// TIA Portal project "水塔水池控制" (V15.1)

(* hardware
DEVICE "S7-1200 station_1"  S7-1200 Station
   slot 0: "Rack_0"  S7-1200 Rack  Rack  V1.0
   slot 1: "PLC_1"  CPU 1214C DC/DC/Rly  6ES7 214-1HG40-0XB0  V4.2
DEVICE "HMI_1"  KTP900 Basic PN
   slot 0: "HMI_1"  KTP900 Basic PN  6AV2 123-2JB03-0AX0  15.1.0.0
   slot 1: "HMI_RT_1"  KTP900 Basic PN  6AV2 123-2JB03-0AX0  15.1.0.0
   slot 5: "HMI_1.IE_CP_1"  PROFINET Interface  15.0.1.0
      slot 1: "PROFINET Interface_1"  PROFINET Interface
         slot 1: "Port_1"  Port
*)

// ===== PLC "PLC_1"  CPU 1214C DC/DC/Rly =====

VAR_GLOBAL   // PLC tag table "默认变量表"
   "S1" AT %M10.0 : Bool;   // 水池下限液位开关
   "S2" AT %M10.1 : Bool;   // 水池上限液位开关
   "S3" AT %M10.2 : Bool;   // 水塔下限液位开关
   "S4" AT %M10.3 : Bool;   // 水塔上限液位开关
   "Start" AT %M10.4 : Bool;
   "Stop" AT %M10.5 : Bool;
   "System_Byte" AT %MB1 : Byte;
   "FirstScan" AT %M1.0 : Bool;
   "DiagStatusUpdate" AT %M1.1 : Bool;
   "AlwaysTRUE" AT %M1.2 : Bool;
   "AlwaysFALSE" AT %M1.3 : Bool;
   "Clock_Byte" AT %MB0 : Byte;
   "Clock_10Hz" AT %M0.0 : Bool;
   "Clock_5Hz" AT %M0.1 : Bool;
   "Clock_2.5Hz" AT %M0.2 : Bool;
   "Clock_2Hz" AT %M0.3 : Bool;
   "Clock_1.25Hz" AT %M0.4 : Bool;
   "Clock_1Hz" AT %M0.5 : Bool;
   "Clock_0.625Hz" AT %M0.6 : Bool;
   "Clock_0.5Hz" AT %M0.7 : Bool;
   "状态0" AT %M2.0 : Bool;
   "状态1" AT %M2.1 : Bool;
   "状态2" AT %M2.2 : Bool;
   "状态3" AT %M2.3 : Bool;
   "状态4" AT %M2.4 : Bool;
   "系统运行状态" AT %M5.0 : Bool;
   "状态5" AT %M2.5 : Bool;
   "Valve" AT %Q0.0 : Bool;
   "Pump" AT %Q0.1 : Bool;
   "Warning" AT %Q0.2 : Bool;
   "水塔状态0" AT %M3.0 : Bool;
   "水塔状态1" AT %M3.1 : Bool;
   "水塔状态2" AT %M3.2 : Bool;
   "水塔状态3" AT %M3.3 : Bool;
   "放水阀" AT %M5.1 : Bool;
   "Byte2" AT %MB2 : Byte;
   "模式选择开关" AT %M5.2 : Bool;
   "Byte3" AT %MB3 : Byte;
   "Tag_1" AT %M5.3 : Bool;
   "手动开阀" AT %M6.0 : Bool;
   "手动启动水泵" AT %M6.1 : Bool;
END_VAR

DATA_BLOCK "HMIdata"   // DB1
{ S7_Optimized_Access := 'TRUE' }
VERSION : 0.1
   VAR
      Tower_water : Int;
      Pool_water : Int;
      Valve_Flow_Num : Int := 10;   // 电磁阀开度
      Pump_Flow_Num : Int := 8;   // 抽水流量大小
      放水阀开度 : Int := 7;   // 放水流量大小
   END_VAR
BEGIN
END_DATA_BLOCK

DATA_BLOCK "水池自动控制_DB"   // DB2
{ S7_Optimized_Access := 'TRUE' }
VERSION : 0.1
// stored: InstanceOfName 水池自动控制
"水池自动控制"
BEGIN
END_DATA_BLOCK

DATA_BLOCK "动画控制_DB"   // DB3
{ S7_Optimized_Access := 'TRUE' }
VERSION : 0.1
// stored: InstanceOfName 动画控制
"动画控制"
BEGIN
END_DATA_BLOCK

DATA_BLOCK "水塔自动控制_DB"   // DB4
{ S7_Optimized_Access := 'TRUE' }
VERSION : 0.1
// stored: InstanceOfName 水塔自动控制
"水塔自动控制"
BEGIN
END_DATA_BLOCK

DATA_BLOCK "手动控制_DB"   // DB5
{ S7_Optimized_Access := 'TRUE' }
VERSION : 0.1
// stored: InstanceOfName 手动控制
"手动控制"
BEGIN
END_DATA_BLOCK

FUNCTION_BLOCK "水池自动控制"   // FB1, LAD
{ S7_Optimized_Access := 'TRUE' }
VERSION : 0.1
   VAR
      T1 : IEC_TIMER;
   END_VAR
   VAR_TEMP   // added for the SCL form of the ladder/FBD networks
      _w1 : Bool;
   END_VAR
BEGIN

REGION Network 1: 初始化
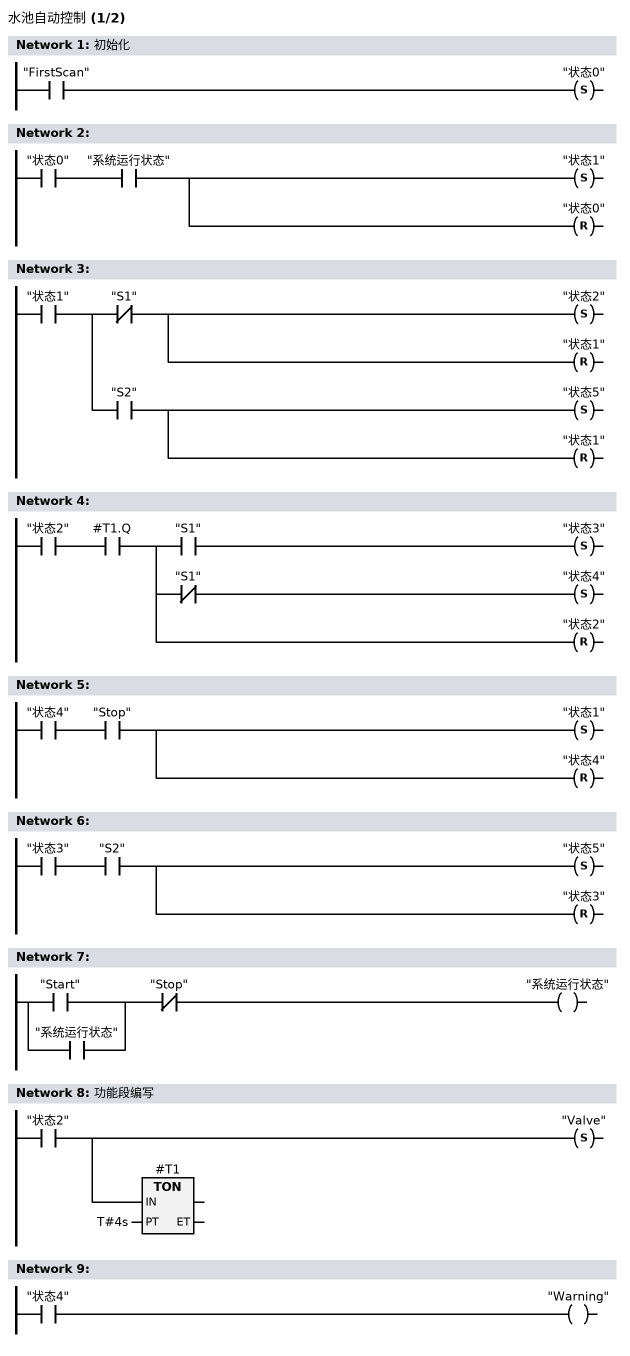
   RUNG wire#powerrail
      Contact( "FirstScan" )
      S_Coil( "状态0" )
   END_RUNG
   // the same network as SCL:
   IF "FirstScan" THEN "状态0" := TRUE; END_IF;
END_REGION

REGION Network 2
   RUNG wire#powerrail
      Contact( "状态0" )
      Contact( "系统运行状态" )
      wire#w1
      S_Coil( "状态1" )
   END_RUNG
   RUNG wire#w1
      R_Coil( "状态0" )
   END_RUNG
   // the same network as SCL:
   IF "状态0" AND "系统运行状态" THEN
       "状态1" := TRUE;
       "状态0" := FALSE;
   END_IF;
END_REGION

REGION Network 3
   RUNG wire#powerrail
      Contact( "状态1" )
      wire#w1
      I_Contact( "S1" )
      wire#w2
      S_Coil( "状态2" )
   END_RUNG
   RUNG wire#w2
      R_Coil( "状态1" )
   END_RUNG
   RUNG wire#w1
      Contact( "S2" )
      wire#w3
      S_Coil( "状态5" )
   END_RUNG
   RUNG wire#w3
      R_Coil( "状态1" )
   END_RUNG
   // the same network as SCL:
   IF "状态1" AND NOT "S1" THEN "状态2" := TRUE; END_IF;
   #_w1 := "状态1";
   IF "状态1" AND NOT "S1" THEN "状态1" := FALSE; END_IF;
   IF #_w1 AND "S2" THEN
       "状态5" := TRUE;
       "状态1" := FALSE;
   END_IF;
END_REGION

REGION Network 4
   RUNG wire#powerrail
      Contact( "状态2" )
      Contact( #T1.Q )
      wire#w1
      Contact( "S1" )
      S_Coil( "状态3" )
   END_RUNG
   RUNG wire#w1
      I_Contact( "S1" )
      S_Coil( "状态4" )
   END_RUNG
   RUNG wire#w1
      R_Coil( "状态2" )
   END_RUNG
   // the same network as SCL:
   #_w1 := "状态2" AND #T1.Q;
   IF #_w1 AND "S1" THEN "状态3" := TRUE; END_IF;
   IF #_w1 AND NOT "S1" THEN "状态4" := TRUE; END_IF;
   IF #_w1 THEN "状态2" := FALSE; END_IF;
END_REGION

REGION Network 5
   RUNG wire#powerrail
      Contact( "状态4" )
      Contact( "Stop" )
      wire#w1
      S_Coil( "状态1" )
   END_RUNG
   RUNG wire#w1
      R_Coil( "状态4" )
   END_RUNG
   // the same network as SCL:
   IF "状态4" AND "Stop" THEN
       "状态1" := TRUE;
       "状态4" := FALSE;
   END_IF;
END_REGION

REGION Network 6
   RUNG wire#powerrail
      Contact( "状态3" )
      Contact( "S2" )
      wire#w1
      S_Coil( "状态5" )
   END_RUNG
   RUNG wire#w1
      R_Coil( "状态3" )
   END_RUNG
   // the same network as SCL:
   IF "状态3" AND "S2" THEN
       "状态5" := TRUE;
       "状态3" := FALSE;
   END_IF;
END_REGION

REGION Network 7
   RUNG wire#powerrail
      Contact( "Start" )
      wire#w1
      I_Contact( "Stop" )
      Coil( "系统运行状态" )
   END_RUNG
   RUNG wire#powerrail
      Contact( "系统运行状态" )
   END_RUNG wire#w1
   // the same network as SCL:
   "系统运行状态" := ("Start" OR "系统运行状态") AND NOT "Stop";
END_REGION

REGION Network 8: 功能段编写
   IF "状态2" THEN "Valve" := TRUE; END_IF;
   #T1.TON(IN := "状态2", PT := T#4s);
END_REGION

REGION Network 9
   RUNG wire#powerrail
      Contact( "状态4" )
      Coil( "Warning" )
   END_RUNG
   // the same network as SCL:
   "Warning" := "状态4";
END_REGION

REGION Network 10
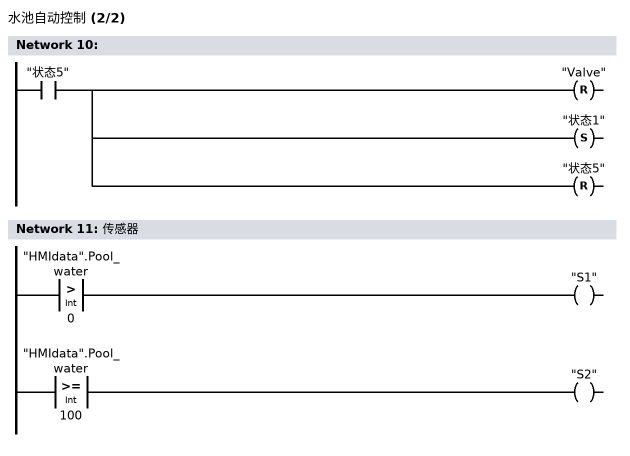
   RUNG wire#powerrail
      Contact( "状态5" )
      wire#w1
      R_Coil( "Valve" )
   END_RUNG
   RUNG wire#w1
      S_Coil( "状态1" )
   END_RUNG
   RUNG wire#w1
      R_Coil( "状态5" )
   END_RUNG
   // the same network as SCL:
   IF "状态5" THEN
       "Valve" := FALSE;
       "状态1" := TRUE;
       "状态5" := FALSE;
   END_IF;
END_REGION

REGION Network 11: 传感器
   RUNG wire#powerrail
      { S7_Templates := "SrcType := Int" } GT_Contact(in1 := "HMIdata".Pool_water, in2 := 0)
      Coil( "S1" )
   END_RUNG
   RUNG wire#powerrail
      { S7_Templates := "SrcType := Int" } GE_Contact(in1 := "HMIdata".Pool_water, in2 := 100)
      Coil( "S2" )
   END_RUNG
   // the same network as SCL:
   "S1" := "HMIdata".Pool_water > 0;
   "S2" := "HMIdata".Pool_water >= 100;
END_REGION
END_FUNCTION_BLOCK

FUNCTION_BLOCK "水塔自动控制"   // FB2, LAD
{ S7_Optimized_Access := 'TRUE' }
VERSION : 0.1
BEGIN

REGION Network 1
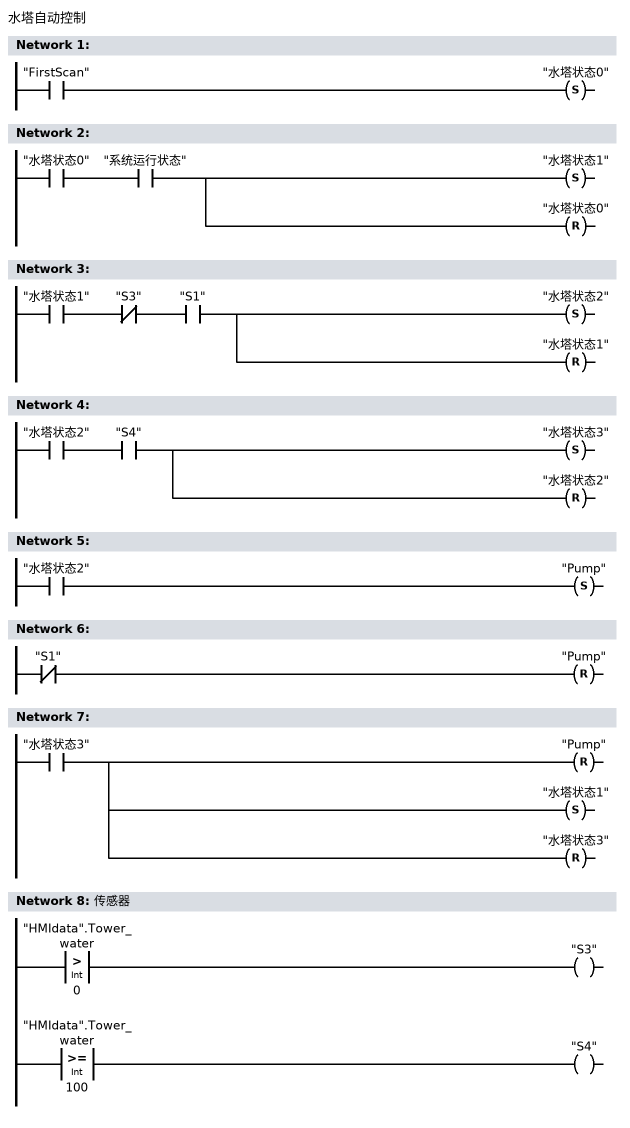
   RUNG wire#powerrail
      Contact( "FirstScan" )
      S_Coil( "水塔状态0" )
   END_RUNG
   // the same network as SCL:
   IF "FirstScan" THEN "水塔状态0" := TRUE; END_IF;
END_REGION

REGION Network 2
   RUNG wire#powerrail
      Contact( "水塔状态0" )
      Contact( "系统运行状态" )
      wire#w1
      S_Coil( "水塔状态1" )
   END_RUNG
   RUNG wire#w1
      R_Coil( "水塔状态0" )
   END_RUNG
   // the same network as SCL:
   IF "水塔状态0" AND "系统运行状态" THEN
       "水塔状态1" := TRUE;
       "水塔状态0" := FALSE;
   END_IF;
END_REGION

REGION Network 3
   RUNG wire#powerrail
      Contact( "水塔状态1" )
      I_Contact( "S3" )
      Contact( "S1" )
      wire#w1
      S_Coil( "水塔状态2" )
   END_RUNG
   RUNG wire#w1
      R_Coil( "水塔状态1" )
   END_RUNG
   // the same network as SCL:
   IF "水塔状态1" AND NOT "S3" AND "S1" THEN
       "水塔状态2" := TRUE;
       "水塔状态1" := FALSE;
   END_IF;
END_REGION

REGION Network 4
   RUNG wire#powerrail
      Contact( "水塔状态2" )
      Contact( "S4" )
      wire#w1
      S_Coil( "水塔状态3" )
   END_RUNG
   RUNG wire#w1
      R_Coil( "水塔状态2" )
   END_RUNG
   // the same network as SCL:
   IF "水塔状态2" AND "S4" THEN
       "水塔状态3" := TRUE;
       "水塔状态2" := FALSE;
   END_IF;
END_REGION

REGION Network 5
   RUNG wire#powerrail
      Contact( "水塔状态2" )
      S_Coil( "Pump" )
   END_RUNG
   // the same network as SCL:
   IF "水塔状态2" THEN "Pump" := TRUE; END_IF;
END_REGION

REGION Network 6
   RUNG wire#powerrail
      I_Contact( "S1" )
      R_Coil( "Pump" )
   END_RUNG
   // the same network as SCL:
   IF NOT "S1" THEN "Pump" := FALSE; END_IF;
END_REGION

REGION Network 7
   RUNG wire#powerrail
      Contact( "水塔状态3" )
      wire#w1
      R_Coil( "Pump" )
   END_RUNG
   RUNG wire#w1
      S_Coil( "水塔状态1" )
   END_RUNG
   RUNG wire#w1
      R_Coil( "水塔状态3" )
   END_RUNG
   // the same network as SCL:
   IF "水塔状态3" THEN
       "Pump" := FALSE;
       "水塔状态1" := TRUE;
       "水塔状态3" := FALSE;
   END_IF;
END_REGION

REGION Network 8: 传感器
   RUNG wire#powerrail
      { S7_Templates := "SrcType := Int" } GT_Contact(in1 := "HMIdata".Tower_water, in2 := 0)
      Coil( "S3" )
   END_RUNG
   RUNG wire#powerrail
      { S7_Templates := "SrcType := Int" } GE_Contact(in1 := "HMIdata".Tower_water, in2 := 100)
      Coil( "S4" )
   END_RUNG
   // the same network as SCL:
   "S3" := "HMIdata".Tower_water > 0;
   "S4" := "HMIdata".Tower_water >= 100;
END_REGION
END_FUNCTION_BLOCK

FUNCTION_BLOCK "动画控制"   // FB3, LAD
{ S7_Optimized_Access := 'TRUE' }
VERSION : 0.1
   VAR
      C1 : IEC_COUNTER;
   END_VAR
   VAR RETAIN
      p1 : Bool;
   END_VAR
   VAR
      p2 : Bool;
      p3 : Bool;
      p4 : Int;
      p5 : Int;
   END_VAR
   VAR_TEMP
      valve_add : Int;   // 电磁阀的注水量
      pump_add : Int;   // 水泵的抽水量
   END_VAR
   VAR_TEMP   // added for the SCL form of the ladder/FBD networks
      _w1 : Bool;
   END_VAR
BEGIN

REGION Network 1: 水池注水控制
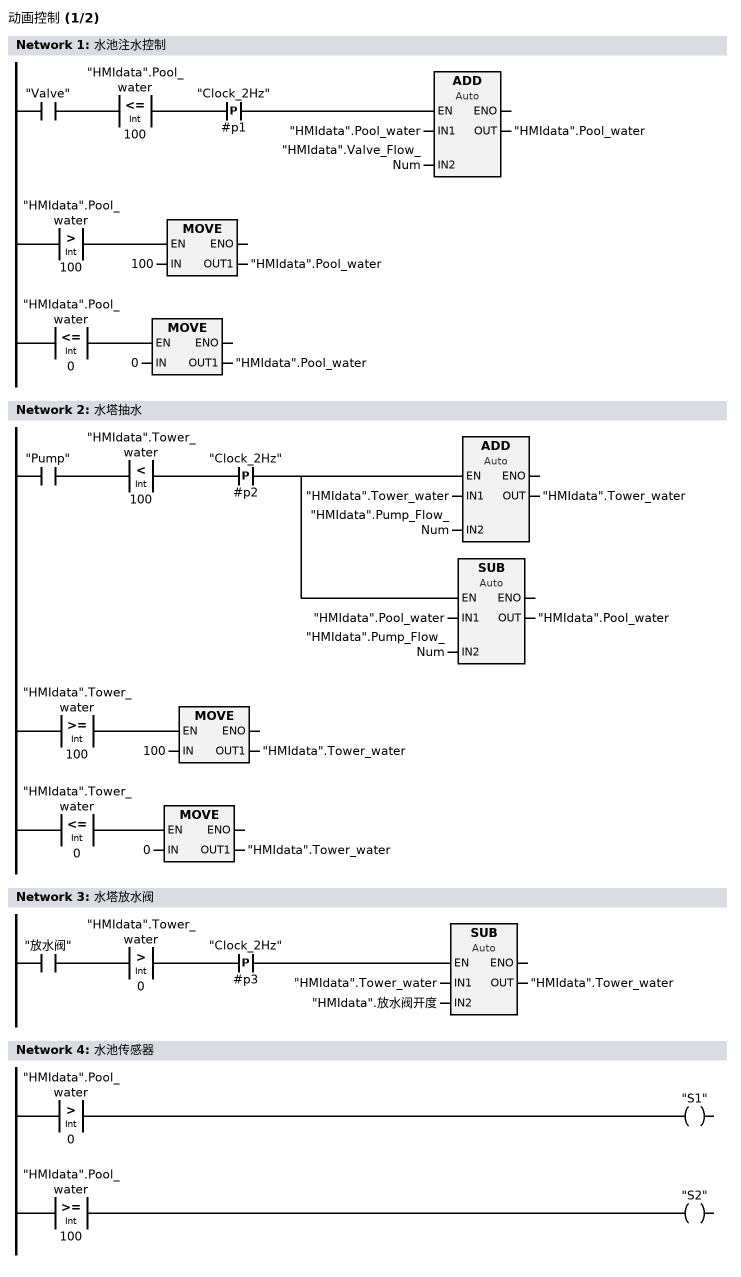
   RUNG wire#powerrail
      Contact( "Valve" )
      { S7_Templates := "SrcType := Int" } LE_Contact(in1 := "HMIdata".Pool_water, in2 := 100)
      P_Contact(operand := "Clock_2Hz", bit := #p1)
      Add(in1 := "HMIdata".Pool_water, in2 := "HMIdata".Valve_Flow_Num, out => "HMIdata".Pool_water)
   END_RUNG
   RUNG wire#powerrail
      { S7_Templates := "SrcType := Int" } GT_Contact(in1 := "HMIdata".Pool_water, in2 := 100)
      Move(in := 100, out1 => "HMIdata".Pool_water)
   END_RUNG
   RUNG wire#powerrail
      { S7_Templates := "SrcType := Int" } LE_Contact(in1 := "HMIdata".Pool_water, in2 := 0)
      Move(in := 0, out1 => "HMIdata".Pool_water)
   END_RUNG
   // the same network as SCL:
   #_w1 := "Valve" AND ("HMIdata".Pool_water <= 100) AND "Clock_2Hz" AND NOT #p1;   // rising edge of "Clock_2Hz"
   #p1 := "Clock_2Hz";
   IF #_w1 THEN "HMIdata".Pool_water := "HMIdata".Pool_water + "HMIdata".Valve_Flow_Num; END_IF;
   IF "HMIdata".Pool_water > 100 THEN "HMIdata".Pool_water := 100; END_IF;
   IF "HMIdata".Pool_water <= 0 THEN "HMIdata".Pool_water := 0; END_IF;
END_REGION

REGION Network 2: 水塔抽水
   RUNG wire#powerrail
      Contact( "Pump" )
      { S7_Templates := "SrcType := Int" } LT_Contact(in1 := "HMIdata".Tower_water, in2 := 100)
      P_Contact(operand := "Clock_2Hz", bit := #p2)
      wire#w1
      Add(in1 := "HMIdata".Tower_water, in2 := "HMIdata".Pump_Flow_Num, out => "HMIdata".Tower_water)
   END_RUNG
   RUNG wire#w1
      Sub(in1 := "HMIdata".Pool_water, in2 := "HMIdata".Pump_Flow_Num, out => "HMIdata".Pool_water)
   END_RUNG
   RUNG wire#powerrail
      { S7_Templates := "SrcType := Int" } GE_Contact(in1 := "HMIdata".Tower_water, in2 := 100)
      Move(in := 100, out1 => "HMIdata".Tower_water)
   END_RUNG
   RUNG wire#powerrail
      { S7_Templates := "SrcType := Int" } LE_Contact(in1 := "HMIdata".Tower_water, in2 := 0)
      Move(in := 0, out1 => "HMIdata".Tower_water)
   END_RUNG
   // the same network as SCL:
   #_w1 := "Pump" AND ("HMIdata".Tower_water < 100) AND "Clock_2Hz" AND NOT #p2;   // rising edge of "Clock_2Hz"
   #p2 := "Clock_2Hz";
   IF #_w1 THEN
       "HMIdata".Tower_water := "HMIdata".Tower_water + "HMIdata".Pump_Flow_Num;
       "HMIdata".Pool_water := "HMIdata".Pool_water - "HMIdata".Pump_Flow_Num;
   END_IF;
   IF "HMIdata".Tower_water >= 100 THEN "HMIdata".Tower_water := 100; END_IF;
   IF "HMIdata".Tower_water <= 0 THEN "HMIdata".Tower_water := 0; END_IF;
END_REGION

REGION Network 3: 水塔放水阀
   RUNG wire#powerrail
      Contact( "放水阀" )
      { S7_Templates := "SrcType := Int" } GT_Contact(in1 := "HMIdata".Tower_water, in2 := 0)
      P_Contact(operand := "Clock_2Hz", bit := #p3)
      Sub(in1 := "HMIdata".Tower_water, in2 := "HMIdata".放水阀开度, out => "HMIdata".Tower_water)
   END_RUNG
   // the same network as SCL:
   #_w1 := "放水阀" AND ("HMIdata".Tower_water > 0) AND "Clock_2Hz" AND NOT #p3;   // rising edge of "Clock_2Hz"
   #p3 := "Clock_2Hz";
   IF #_w1 THEN "HMIdata".Tower_water := "HMIdata".Tower_water - "HMIdata".放水阀开度; END_IF;
END_REGION

REGION Network 4: 水池传感器
   RUNG wire#powerrail
      { S7_Templates := "SrcType := Int" } GT_Contact(in1 := "HMIdata".Pool_water, in2 := 0)
      Coil( "S1" )
   END_RUNG
   RUNG wire#powerrail
      { S7_Templates := "SrcType := Int" } GE_Contact(in1 := "HMIdata".Pool_water, in2 := 100)
      Coil( "S2" )
   END_RUNG
   // the same network as SCL:
   "S1" := "HMIdata".Pool_water > 0;
   "S2" := "HMIdata".Pool_water >= 100;
END_REGION

REGION Network 5: 水塔传感器
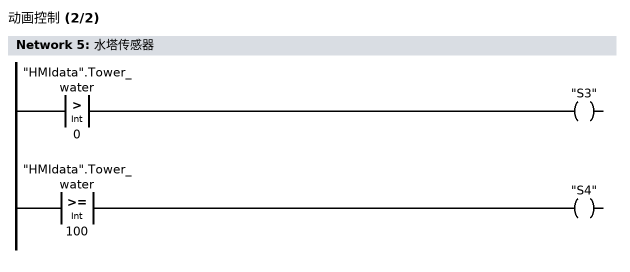
   RUNG wire#powerrail
      { S7_Templates := "SrcType := Int" } GT_Contact(in1 := "HMIdata".Tower_water, in2 := 0)
      Coil( "S3" )
   END_RUNG
   RUNG wire#powerrail
      { S7_Templates := "SrcType := Int" } GE_Contact(in1 := "HMIdata".Tower_water, in2 := 100)
      Coil( "S4" )
   END_RUNG
   // the same network as SCL:
   "S3" := "HMIdata".Tower_water > 0;
   "S4" := "HMIdata".Tower_water >= 100;
END_REGION
END_FUNCTION_BLOCK

FUNCTION_BLOCK "手动控制"   // FB4, LAD
{ S7_Optimized_Access := 'TRUE' }
VERSION : 0.1
BEGIN

REGION Network 1
   // 水池水位未达到高液位时，手动打开电磁阀
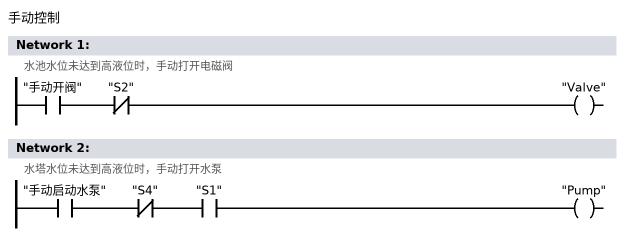
   RUNG wire#powerrail
      Contact( "手动开阀" )
      I_Contact( "S2" )
      Coil( "Valve" )
   END_RUNG
   // the same network as SCL:
   "Valve" := "手动开阀" AND NOT "S2";
END_REGION

REGION Network 2
   // 水塔水位未达到高液位时，手动打开水泵
   RUNG wire#powerrail
      Contact( "手动启动水泵" )
      I_Contact( "S4" )
      Contact( "S1" )
      Coil( "Pump" )
   END_RUNG
   // the same network as SCL:
   "Pump" := "手动启动水泵" AND NOT "S4" AND "S1";
END_REGION
END_FUNCTION_BLOCK

FUNCTION "模式选择" : Void   // FC1, LAD
{ S7_Optimized_Access := 'TRUE' }
VERSION : 0.1
BEGIN

REGION Network 1: "模式选择开关":0-手动模式 1-自动模式
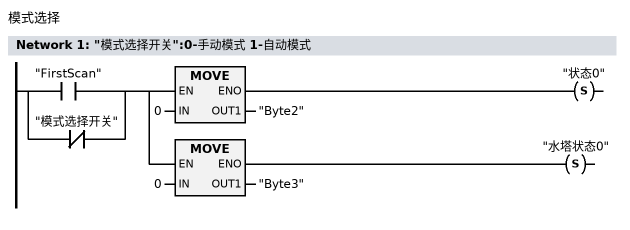
   RUNG wire#powerrail
      Contact( "FirstScan" )
      wire#w1
      Move(in := 0, out1 => "Byte2")
      S_Coil( "状态0" )
   END_RUNG
   RUNG wire#powerrail
      I_Contact( "模式选择开关" )
   END_RUNG wire#w1
   RUNG wire#w1
      Move(in := 0, out1 => "Byte3")
      S_Coil( "水塔状态0" )
   END_RUNG
   // the same network as SCL:
   IF "FirstScan" OR NOT "模式选择开关" THEN
       "Byte2" := 0;
       "状态0" := TRUE;
       "Byte3" := 0;
       "水塔状态0" := TRUE;
   END_IF;
END_REGION
END_FUNCTION

ORGANIZATION_BLOCK "Main"   // OB1, LAD, ProgramCycle
TITLE = "Main Program Sweep (Cycle)"
{ S7_Optimized_Access := 'TRUE' }
VERSION : 0.1
   VAR_INPUT
      Initial_Call : Bool;   // Initial call of this OB
      Remanence : Bool;   // =True, if remanent data are available
   END_VAR
   VAR_TEMP   // added for the SCL form of the ladder/FBD networks
      _w1 : Bool;
   END_VAR
BEGIN

REGION Network 1
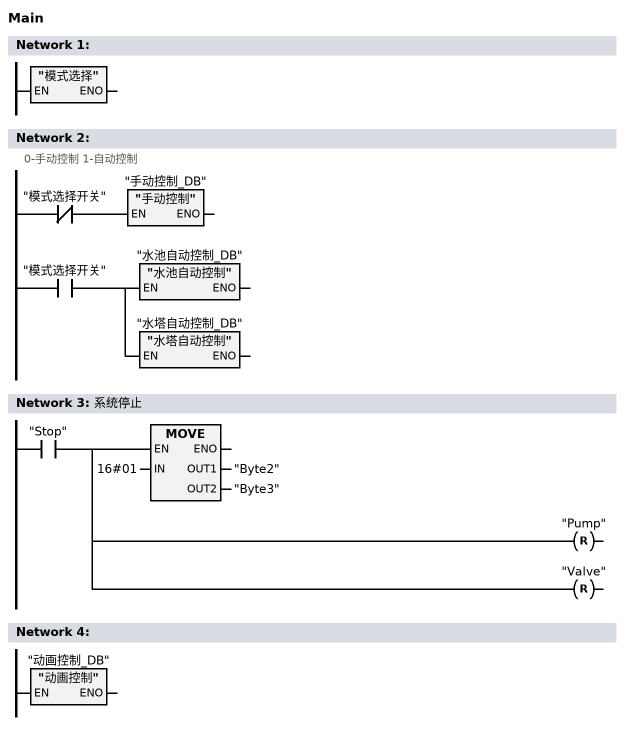
   RUNG wire#powerrail
      "模式选择"()
   END_RUNG
   // the same network as SCL:
   "模式选择"();
END_REGION

REGION Network 2
   // 0-手动控制 1-自动控制
   RUNG wire#powerrail
      I_Contact( "模式选择开关" )
      "手动控制_DB"()
   END_RUNG
   RUNG wire#powerrail
      Contact( "模式选择开关" )
      wire#w1
      "水池自动控制_DB"()
   END_RUNG
   RUNG wire#w1
      "水塔自动控制_DB"()
   END_RUNG
   // the same network as SCL:
   IF NOT "模式选择开关" THEN
       "手动控制_DB"();   // "手动控制"
   END_IF;
   #_w1 := "模式选择开关";
   IF #_w1 THEN
       "水池自动控制_DB"();   // "水池自动控制"
       "水塔自动控制_DB"();   // "水塔自动控制"
   END_IF;
END_REGION

REGION Network 3: 系统停止
   RUNG wire#powerrail
      Contact( "Stop" )
      wire#w1
      Move(in := 16#01, out1 => "Byte2", out2 => "Byte3")
   END_RUNG
   RUNG wire#w1
      R_Coil( "Pump" )
   END_RUNG
   RUNG wire#w1
      R_Coil( "Valve" )
   END_RUNG
   // the same network as SCL:
   IF "Stop" THEN
       "Byte2" := 16#01;
       "Byte3" := 16#01;
       "Pump" := FALSE;
       "Valve" := FALSE;
   END_IF;
END_REGION

REGION Network 4
   RUNG wire#powerrail
      "动画控制_DB"()
   END_RUNG
   // the same network as SCL:
   "动画控制_DB"();   // "动画控制"
END_REGION
END_ORGANIZATION_BLOCK

(* ===== HMI "HMI_RT_1" =====
system functions are stored by id; their names below are inferred from use
connection "HMI_连接_1": ETHERNET, SMART_S7_1200_OMS

HMI tags "默认变量表"
   "HMIdata_Tower_water" : Int = PLC HMIdata.Tower_water, 100 ms
   "HMIdata_Pool_water" : Int = PLC HMIdata.Pool_water, 100 ms
   "Start" : Bool = PLC Start AT %M10.4, 100 ms
   "Stop" : Bool = PLC Stop AT %M10.5, 100 ms
   "放水阀" : Bool = PLC 放水阀 AT %M5.1, 100 ms
   "Pump" : Bool = PLC Pump AT %Q0.1, 100 ms
   "Valve" : Bool = PLC Valve AT %Q0.0, 100 ms
   "Warning" : Bool = PLC Warning AT %Q0.2, 100 ms
   "S1" : Bool = PLC S1 AT %M10.0, 100 ms
   "S2" : Bool = PLC S2 AT %M10.1, 100 ms
   "S4" : Bool = PLC S4 AT %M10.3, 100 ms
   "S3" : Bool = PLC S3 AT %M10.2, 100 ms
   "HMIdata_Pump_Flow_Num" : Int = PLC HMIdata.Pump_Flow_Num, 100 ms
   "HMIdata_放水阀开度" : Int = PLC HMIdata.放水阀开度, 100 ms
   "HMIdata_Valve_Flow_Num" : Int = PLC HMIdata.Valve_Flow_Num, 100 ms
   "模式选择开关" : Bool = PLC 模式选择开关 AT %M5.2, 100 ms
   "手动启动水泵" : Bool = PLC 手动启动水泵 AT %M6.1, 1 s
   "手动开阀" : Bool = PLC 手动开阀 AT %M6.0, 1 s
   "系统运行状态" : Bool = PLC 系统运行状态 AT %M5.0, 1 s

text list "阀门开度": 1 '开度：1'; 2 '开度：2'; 3 '开度：3'; 4 '开度：4'; 5 '开度：5'; 6 '开度：6'; 7 '开度：7'; 8 '开度：8'; 9 '开度：9'; 10 '开度：10'

screen "主菜单" 800x480
   Button "按钮_1" at 684,254 size 96x32; TextOff '启动'
      on Press: SetBit("Start")
      on Release: ResetBit("Start")
      Appearance <- "系统运行状态"
   Button "按钮_2" at 684,298 size 96x32; TextOff '停止'
      on Press: SetBit("Stop")
      on Release: ResetBit("Stop")
   Circle "圆_2" at 582,11 size 45x45
      Appearance <- "Pump"
   Circle "圆_3" at 646,11 size 45x45
      Appearance <- "Valve"
   Circle "圆_4" at 701,11 size 45x45
      Appearance <- "Warning"
   TextField "文本域_2" at 582,65 size 41x21; Text '抽水'
   TextField "文本域_3" at 633,65 size 59x21; Text '电磁阀'
   TextField "文本域_4" at 701,65 size 41x21; Text '故障'
   Group "Group_1" at 514,365 size 111x49; Picture "图形_14"
   Group "Group_2" at 514,271 size 111x49; Picture "图形_14"
   Group "Group_3" at 205,173 size 111x49; Picture "图形_14"
   Group "Group_4" at 205,46 size 111x49; Picture "图形_14"
   Bar "棒图_1" at 112,60 size 127x150; MinimumValue 0; MaximumValue 100
      ProcessValue <- "HMIdata_Tower_water"
   Bar "棒图_2" at 353,289 size 192x111; MinimumValue 0; MaximumValue 100
      ProcessValue <- "HMIdata_Pool_water"
   GraphicView "图形视图_11" at 342,54 size 52x103; Picture "图形_18"
   Group "Group_6" at 179,5 size 217x55; Picture "图形_23"
   GraphicView "图形视图_19" at 364,235 size 52x139; Picture "图形_18"
   Group "Group_7" at 352,143 size 70x100; Picture "图形_24"
   Group "Group_8" at 474,145 size 167x55; Picture "图形_19"
   GraphicView "图形视图_20" at 474,198 size 57x105; Picture "图形_18"
   GraphicView "图形视图_23" at 731,149 size 69x47; Picture "图形_20"
   Group "Group_5" at 632,110 size 137x88; Picture "图形_21"
   GraphicView "图形视图_24" at 55,166 size 63x50; Picture "图形_20"
   Group "Group" at 0,161 size 61x44; Picture "图形_13"
   Button "按钮_4" at 82,437 size 192x32; TextOff '水塔管理'; TextOn '水塔管理页面'
      on Click: ActivateScreen("水塔管理页面", 0)
   Button "按钮_5" at 352,437 size 192x32; TextOff '水池管理'
      on Click: ActivateScreen("水池管理", 0)
   Rectangle "矩形_18" at 387,309 size 7x17
      Appearance <- "Pump"
      Visibility <- "Pump"
   Rectangle "矩形_19" at 387,288 size 7x17
      Visibility <- "Pump"
      Appearance <- "Pump"
   Rectangle "矩形_5" at 557,166 size 18x7
      Visibility <- "Valve"
      Appearance <- "Valve"
   Rectangle "矩形_6" at 529,166 size 18x7
      Visibility <- "Valve"
      Appearance <- "Valve"
   Button "按钮_6" at 684,344 size 96x32; TextOff '手动/自动'
      on Click: InvertBit("模式选择开关")
   Circle "圆_5" at 501,11 size 45x45
      Appearance <- "模式选择开关"
   TextField "文本域_5" at 484,64 size 77x21; Text '自动模式'
      Visibility <- "模式选择开关"
   TextField "文本域_6" at 484,65 size 77x21; Text '手动模式'
      Visibility <- "模式选择开关"
   Button "按钮_7" at 684,393 size 96x32; TextOff '启动水泵'
      on Click: InvertBit("手动启动水泵")
      Appearance <- "手动启动水泵"
   Button "按钮_8" at 684,439 size 96x32; TextOff '启动电磁阀'
      on Click: InvertBit("手动开阀")
      Appearance <- "手动开阀"
   Button "按钮_3" at 10,227 size 79x27; TextOff '放水阀'
      on Click: InvertBit("放水阀")
      Appearance <- "放水阀"
   Rectangle "矩形_8" at 387,265 size 7x17
      Visibility <- "Pump"
      Appearance <- "Pump"
   Rectangle "矩形_9" at 387,244 size 7x17
      Visibility <- "Pump"
      Appearance <- "Pump"
   Rectangle "矩形_10" at 387,354 size 7x17
      Visibility <- "Pump"
      Appearance <- "Pump"
   Rectangle "矩形_11" at 387,333 size 7x17
      Visibility <- "Pump"
      Appearance <- "Pump"
   Rectangle "矩形_13" at 364,124 size 7x17
      Visibility <- "Pump"
      Appearance <- "Pump"
   Rectangle "矩形_20" at 364,103 size 7x17
      Visibility <- "Pump"
      Appearance <- "Pump"
   Rectangle "矩形_14" at 364,80 size 7x17
      Visibility <- "Pump"
      Appearance <- "Pump"
   Rectangle "矩形_15" at 364,59 size 7x17
      Visibility <- "Pump"
      Appearance <- "Pump"
   Rectangle "矩形_22" at 251,28 size 17x7
      Visibility <- "Pump"
      Appearance <- "Pump"
   Rectangle "矩形_23" at 228,28 size 17x7
      Visibility <- "Pump"
      Appearance <- "Pump"
   Rectangle "矩形_24" at 298,28 size 17x7
      Visibility <- "Pump"
      Appearance <- "Pump"
   Rectangle "矩形_25" at 275,28 size 17x7
      Visibility <- "Pump"
      Appearance <- "Pump"
   Rectangle "矩形_27" at 322,28 size 17x7
      Visibility <- "Pump"
      Appearance <- "Pump"
   Rectangle "矩形_1" at 501,257 size 7x18
      Visibility <- "Valve"
      Appearance <- "Valve"
   Rectangle "矩形_7" at 501,281 size 7x18
      Visibility <- "Valve"
      Appearance <- "Valve"
   Rectangle "矩形_12" at 501,209 size 7x18
      Visibility <- "Valve"
      Appearance <- "Valve"
   Rectangle "矩形_21" at 501,233 size 7x18
      Visibility <- "Valve"
      Appearance <- "Valve"
   Rectangle "矩形_2" at 613,167 size 18x7
      Visibility <- "Valve"
      Appearance <- "Valve"
   Rectangle "矩形_3" at 585,167 size 18x7
      Visibility <- "Valve"
      Appearance <- "Valve"
   GraphicView "图形视图_1" at 1,161 size 60x44; Picture "图形_13"
      Visibility <- "放水阀"
   GraphicView "图形视图_2" at 0,161 size 60x44; Picture "图形_10"
      Visibility <- "放水阀"
   GraphicView "图形视图_8" at 514,365 size 111x49; Picture "图形_14"
      Visibility <- "S1"
   GraphicView "图形视图_7" at 514,365 size 111x49; Picture "图形_16"
      Visibility <- "S1"
   GraphicView "图形视图_3" at 514,271 size 111x49; Picture "图形_14"
      Visibility <- "S2"
   GraphicView "图形视图_4" at 514,271 size 111x49; Picture "图形_16"
      Visibility <- "S2"
   GraphicView "图形视图_5" at 205,173 size 111x49; Picture "图形_14"
      Visibility <- "S3"
   GraphicView "图形视图_6" at 205,173 size 111x49; Picture "图形_16"
      Visibility <- "S3"
   GraphicView "图形视图_9" at 205,46 size 111x49; Picture "图形_14"
      Visibility <- "S4"
   GraphicView "图形视图_10" at 205,46 size 111x49; Picture "图形_16"
      Visibility <- "S4"
   GraphicView "图形视图_14" at 632,110 size 137x88; Picture "图形_21"
      Visibility <- "Valve"
   GraphicView "图形视图_15" at 632,110 size 137x88; Picture "图形_22"
      Visibility <- "Valve"
   GraphicView "图形视图_16" at 340,5 size 56x55; Picture "图形_23"
   GraphicView "图形视图_12" at 179,5 size 58x55; Picture "图形_19"
   GraphicView "图形视图_13" at 232,5 size 114x55; Picture "图形_20"
   GraphicView "图形视图_17" at 352,143 size 70x100; Picture "图形_24"
      Visibility <- "Pump"
   GraphicView "图形视图_18" at 352,143 size 70x100; Picture "图形_25"
      Visibility <- "Pump"
   GraphicView "图形视图_21" at 474,145 size 58x55; Picture "图形_19"
   GraphicView "图形视图_22" at 527,145 size 114x55; Picture "图形_20"

screen "水塔管理页面" 800x480
   Button "按钮_1" at 591,437 size 192x32; TextOff '主菜单'
      on Click: ActivateScreen("主菜单", 0)
   Group "Group_4" at 356,104 size 98x47; Picture "图形_14"
   Group "Group_3" at 336,381 size 118x42; Picture "图形_14"
   Bar "棒图_1" at 218,106 size 167x317; MinimumValue 0; MaximumValue 100
      ProcessValue <- "HMIdata_Tower_water"
   Button "按钮_3" at 99,431 size 100x37; TextOff '放水阀'
      on Click: InvertBit("放水阀")
      Appearance <- "放水阀"
   GraphicView "图形视图_24" at 155,373 size 63x50; Picture "图形_20"
   Group "Group" at 100,368 size 61x44; Picture "图形_13"
   SymbolicIOField "符号 I/O 域_1" at 589,235 size 96x32; TextOff '0'; TextOn '1'; TextList "阀门开度"
      ProcessValue <- "HMIdata_Pump_Flow_Num"
   TextField "文本域_1" at 463,240 size 107x20; Text '抽水流量大小'
   TextField "文本域_2" at 463,291 size 107x20; Text '放水流量大小'
   SymbolicIOField "符号 I/O 域_2" at 589,293 size 96x32; TextOn '1'; TextOff '0'; TextList "阀门开度"
      ProcessValue <- "HMIdata_放水阀开度"
   TextField "文本域_3" at 269,22 size 125x33; Text '水塔控制'
   TextField "文本域_4" at 478,164 size 77x21; Text '当前水位'
   IOField "I/O 域_1" at 587,159 size 99x32; FormatPattern s999999
      ProcessValue <- "HMIdata_Tower_water"
   Button "按钮_7" at 591,368 size 96x32; TextOff '启动水泵'
      on Click: InvertBit("手动启动水泵")
      Appearance <- "手动启动水泵"
   GraphicView "图形视图_9" at 356,104 size 98x47; Picture "图形_14"
      Visibility <- "S4"
   GraphicView "图形视图_10" at 356,104 size 98x47; Picture "图形_16"
      Visibility <- "S4"
   GraphicView "图形视图_5" at 336,381 size 118x42; Picture "图形_14"
      Visibility <- "S3"
   GraphicView "图形视图_6" at 336,381 size 118x42; Picture "图形_16"
      Visibility <- "S3"
   GraphicView "图形视图_1" at 101,368 size 60x44; Picture "图形_13"
      Visibility <- "放水阀"
   GraphicView "图形视图_2" at 100,368 size 60x44; Picture "图形_10"
      Visibility <- "放水阀"

screen "水池管理" 800x480
   GraphicView "图形视图_3" at 337,188 size 111x52; Picture "图形_14"
      Visibility <- "S2"
   GraphicView "图形视图_4" at 337,188 size 111x52; Picture "图形_16"
      Visibility <- "S2"
   GraphicView "图形视图_8" at 335,274 size 111x52; Picture "图形_14"
      Visibility <- "S1"
   GraphicView "图形视图_7" at 335,274 size 111x52; Picture "图形_16"
      Visibility <- "S1"
   Circle "圆_1" at 571,23 size 33x33
      Appearance <- "放水阀"
   Circle "圆_2" at 628,23 size 33x33
      Appearance <- "Pump"
   Circle "圆_3" at 676,23 size 33x33
      Appearance <- "Valve"
   Circle "圆_4" at 727,23 size 33x33
      Appearance <- "Warning"
   TextField "文本域_1" at 551,59 size 59x21; Text '放水阀'
   TextField "文本域_2" at 625,59 size 41x21; Text '抽水'
   TextField "文本域_3" at 666,59 size 59x21; Text '电磁阀'
   TextField "文本域_4" at 728,59 size 41x21; Text '故障'
   Button "按钮_1" at 587,437 size 192x32; TextOff '主菜单'
      on Click: ActivateScreen("主菜单", 0)
   Group "Group_2" at 337,188 size 111x52; Picture "图形_14"
   Group "Group_1" at 335,274 size 111x52; Picture "图形_14"
   Bar "棒图_2" at 181,203 size 192x114; MinimumValue 0; MaximumValue 100
      ProcessValue <- "HMIdata_Pool_water"
   Group "Group" at 551,23 size 218x57
   SymbolicIOField "符号 I/O 域_1" at 589,235 size 96x32; TextOn '1'; TextOff '0'; TextList "阀门开度"
      ProcessValue <- "HMIdata_Valve_Flow_Num"
   TextField "文本域_5" at 463,240 size 124x20; Text '电磁阀流量大小'
   TextField "文本域_7" at 478,164 size 77x21; Text '当前水位'
   IOField "I/O 域_1" at 587,159 size 99x32; FormatPattern s999999
      ProcessValue <- "HMIdata_Pool_water"
   Button "按钮_8" at 585,367 size 117x40; TextOff '启动电磁阀'
      on Click: InvertBit("手动开阀")
      Appearance <- "手动开阀"
   TextField "文本域_6" at 222,44 size 125x33; Text '水池控制'
*)